(* Logix 5000 project; controller cal1615 1756-L62 rev 20.11; software revision 20.05; part 11 of 82 *)
(* tags used below, declared in another part *)
   FAULT : BOOL;   // Fault AFI
   p00_wac : Accumulator;   // Winder Accumulator
   p01_di_edge_ctrl_estop_active : BOOL;   // System Digital Input Edge Control Estop Active
   p01_di_estop_1_tripped : BOOL;   // System Digital Input EStop Relay 1 Tripped
   p01_di_estop_2_tripped : BOOL;   // System Digital Input EStop Relay 2 Tripped
   p01_di_estop_reset : BOOL;   // System Digital Inupt Main Operator Panel E-Stop Reset
   p01_di_impreg_estop_active : BOOL;   // System Digital Input Impreg Estop Active
   p01_di_letoff_estop_active : BOOL;   // System Digital Input Letoff Estop Active
   p01_di_lof_acc_estop_active : BOOL;   // System Digital Input Letoff Accumulator Estop Active
   p01_di_main_hmi_estop : BOOL;   // System Digital Inupt Main Operator Panel E-Stop Active
   p01_di_rope_sw_1_active : BOOL;   // System Digital Input Rope Switch 1 Active
   p01_di_rope_sw_2_active : BOOL;   // System Digital Input Rope Switch 2 Active
   p01_di_rope_sw_3_active : BOOL;   // System Digital Input Rope Switch 3 Active
   p01_di_rope_sw_4_active : BOOL;   // System Digital Input Rope Switch 4 Active
   p01_di_rope_sw_5_active : BOOL;   // System Digital Input Rope Switch 5 Active
   p01_di_rope_sw_6_active : BOOL;   // System Digital Input Rope Switch 6 Active
   p01_di_rope_sw_7_active : BOOL;   // System Digital Input Rope Switch 7 Active
   p01_di_rope_sw_8_active : BOOL;   // System Digital Input Rope Switch 8 Active
   p01_di_splice_estop_active : BOOL;   // System Digital Input Splice Press Estop Active
   p01_di_ts2_estop_active : BOOL;   // System Digital Input Tension Stand 2 Estop Active
   p01_di_winder_estop_active : BOOL;   // System Digital Input Winder Estop Active
   p01_recipe_active : recipe;   // Active Recipe
   p01r01 : routine;
   p01r02_do_buzzer_LINE : BOOL;
   p01r02_do_green_stack_light_lel : BOOL;   // System Outputs Green Stack Light
   p01r02_do_green_stack_light_LINE : BOOL;
   p01r02_do_red_stack_light : BOOL;   // System Outputs Red Stack Light
   p01r02_do_red_stack_light_LINE : BOOL;
   p01r02_do_yellow_stack_light_LINE : BOOL;
   p01r02_fault_exists : BOOL;
   p01r02_timer_second : TIMER[2];   // System Misc Control Timer Second Pulse
   p01r02_unack_fault : BOOL;   // System Misc Control Unacknowledged Fault Exists
   p01r02_unack_warning : BOOL;   // System Misc Control Unacknowledged Warning Exists
   p01r02_warnings_exists : BOOL;
   p01r04 : routine;   // System Outputs
   p01r09 : routine;   // System Modes
   p01r09_estop_ok : BOOL;   // System Modes Estop Dwell OK
   p01r09_mode_run : BOOL;   // System Modes All Modes Run Mode
   p01r09_open_oven : BOOL;
   p01r09_open_oven_toggle : SYS_Toggle;
   p01r09_pb_global_reset : BOOL;   // System Modes PB: Global Fault Reset
   p01r09_pb_line_jog : BOOL;   // System Modes PB: Line Jog Forward
   p01r09_permissive_change : BOOL;   // System Modes Permissive Mode Change
   p01r09_stretch_mode : BOOL;
   p01r09_timer_estop_reset : TIMER;   // System Modes Estop Reset Dwell
   p01r09_timer_fault : TIMER[20];   // System Modes Fault Delay
   p01r09_timer_global_reset : TIMER;   // System Modes Global Reset Timer
   p01r09_timer_warning : TIMER[4];   // System Modes Warning Delay
   p01r10 : routine;   // System Annunciators
   p01r10_fault_exists : BOOL;
   p01r10_unack_fault : DINT;
   p01r10_unack_fault_ex : BOOL;
   p01r10_unack_warn_ex : BOOL;   // System Annunciators Unacknowledged Warning Exists
   p01r10_unack_warning : DINT;   // System Annunciators Unacknowledged Warning Exists
   p01r10_warning_exists : BOOL;
   p01r12_zero_line_speed : BOOL;   // System Line Accel Decel Control Line Speed at Zero
   p01r13_permissive_drives : BOOL;   // System Line Start Sequence Permissive Drives
   p01r13_permissive_line_run : BOOL;   // System Line Start Sequence Permissive Line Run
   p01r13_state : DINT;   // System Line Start Sequence Sequencer Step
   p01r13_status : DINT;   // System Line Start Sequence Encoded Step
   p02_dint_from_hmi : hmi_dint;
   p11r02_fault_exists : BOOL;
   p11r02_unack_fault : BOOL;   // Zone 1 Misc Control Unacknowledged Fault Exists
   p11r02_unack_warning : BOOL;   // Zone 1 Misc Control Unacknowledged Warning Exists
   p11r02_warning_exists : BOOL;
   p11r30 : routine;   // Zone 1 Temperature Control
   p12r02_fault_exists : BOOL;
   p12r02_unack_fault : BOOL;   // Zone 2 Misc Control Unacknowledged Fault Exists
   p12r02_unack_warning : BOOL;   // Zone 2 Misc Control Unacknowledged Warning Exists
   p12r02_warning_exists : BOOL;
   p12r30 : routine;   // Zone 2 Temperature Control
   p13r02_fault_exists : BOOL;
   p13r02_unack_fault : BOOL;   // Zone 3 Misc Control Unacknowledged Fault Exists
   p13r02_unack_warning : BOOL;   // Zone 3 Misc Control Unacknowledged Warning Exists
   p13r02_warning_exists : BOOL;
   p19r02_fault_exists : BOOL;
   p19r02_unack_warning : BOOL;   // Advanced Cooling Misc Control Unacknowledged Warning
   p19r02_warning_exists : BOOL;
   p20r02_fault_exists : BOOL;
   p20r02_unack_fault : BOOL;   // Letoff Misc Control Unacknowledge Fault Exists
   p20r02_unack_warning : BOOL;   // Letoff Misc Control Unacknowledge Warning Exists
   p20r02_warning_exists : BOOL;
   p21r02_fault_exists : BOOL;
   p21r02_unack_fault : BOOL;   // Splice Press Misc Control Unacknowledged Fault Exists
   p21r02_unack_warning : BOOL;   // Splice Press Misc Control Unacknowledged Warning Exists
   p21r02_warning_exists : BOOL;
   p22r02_fault_exists : BOOL;
   p22r02_unack_fault : BOOL;   // Impreg Pickup Roll Misc Control Unacknowledged Fault Exists
   p22r02_unack_warning : BOOL;   // Impreg Pickup Roll Misc Control Unacknowledged Warning Exists
   p22r02_warning_exists : BOOL;
   p22r09_mode_run : BOOL;   // Tension Stand 1 Modes Run Mode
   p23r02 : routine;   // Impreg Misc Control
   p23r02_fault_exists : BOOL;
   p23r02_unack_fault : BOOL;   // Imperg Misc Control Unackn. Fault Exist
   p23r02_unack_warning : BOOL;   // Impreg Misc Control Unackn. Warning Exist
   p23r02_warning_exists : BOOL;
   p24r02_fault_exists : BOOL;
   p24r02_unack_fault : BOOL;   // Tension Stand 2 Misc Control Unacknowledged Fault Exists
   p24r02_unack_warning : BOOL;   // Tension Stand 2 Misc Control Unacknowledged Warning Exists
   p24r02_warning_exists : BOOL;
   p25r02_fault_exists : BOOL;
   p25r02_unack_fault : BOOL;   // Upper Poly Letoff Misc Control Unacknowledged Fault Exists
   p25r02_unack_warning : BOOL;   // Upper Poly Letoff Misc Control Unacknowledged Warning Exists
   p25r02_warning_exists : BOOL;
   p25r09_mode_run : BOOL;   // Tension Stand 2 Modes Run Mode
   p26r02_fault_exists : BOOL;
   p26r02_unack_fault : BOOL;   // Upper Poly Letoff Misc Control Unacknowledged Fault Exists
   p26r02_unack_warning : BOOL;   // Upper Poly Letoff Misc Control Unacknowledged Warning Exists
   p26r02_warning_exists : BOOL;
   p27r02_fault_exists : BOOL;
   p27r02_unack_fault : BOOL;   // Lower Poly Letoff Misc Control Unacknowledged Fault Exists
   p27r02_unack_warning : BOOL;   // Lower Poly Letoff Misc Control Unacknowledged Warning Exists
   p27r02_warning_exists : BOOL;
   p28r02_fault_exists : BOOL;
   p28r02_unack_fault : BOOL;
   p28r02_unack_warning : BOOL;
   p28r02_warning_exists : BOOL;
   p29r02_fault_exists : BOOL;
   p29r02_unack_fault : BOOL;   // Winder Misc Control Unacknowledged Fault Exists
   p29r02_unack_warning : BOOL;   // Winder Misc Control Unackn. Warning Exists
   p29r02_warning_exists : BOOL;
   p30r02_fault_exists : BOOL;
   p30r02_warning_exists : BOOL;
(* P01_System, continued *)

ROUTINE R09_Modes   (* ladder *)
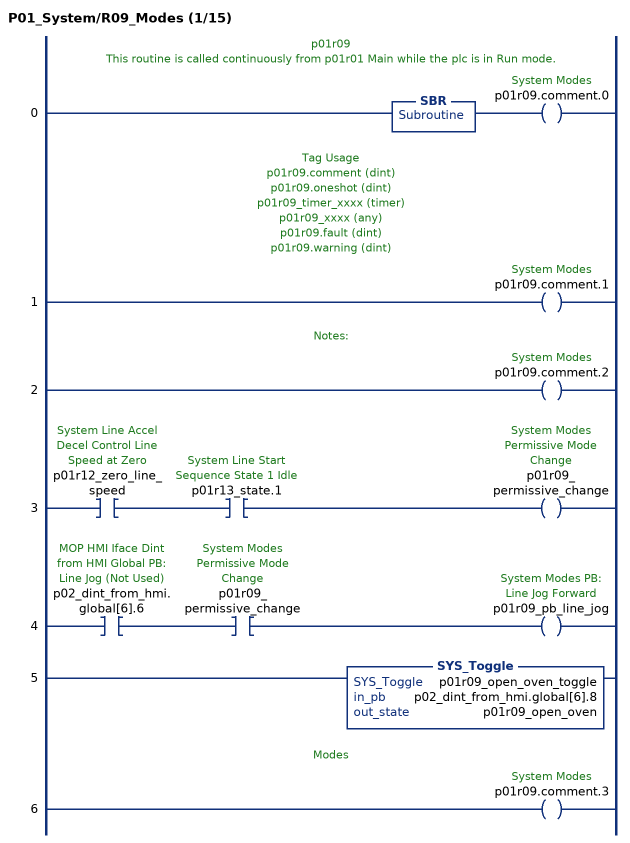
   // p01r09
   // This routine is called continuously from p01r01 Main while the plc is in Run mode.
   0: SBR()OTE(p01r09.comment.0);
   // Tag Usage
   // p01r09.comment (dint)
   // p01r09.oneshot (dint)
   // p01r09_timer_xxxx (timer)
   // p01r09_xxxx (any)
   // p01r09.fault (dint)
   // p01r09.warning (dint)
   1: OTE(p01r09.comment.1);
   // Notes:
   2: OTE(p01r09.comment.2);
   3: XIC(p01r12_zero_line_speed)XIC(p01r13_state.1)OTE(p01r09_permissive_change);
   4: XIC(p02_dint_from_hmi.global[6].6)XIC(p01r09_permissive_change)OTE(p01r09_pb_line_jog);
   5: SYS_Toggle(p01r09_open_oven_toggle,p02_dint_from_hmi.global[6].8,p01r09_open_oven);
   // Modes
   6: OTE(p01r09.comment.3);
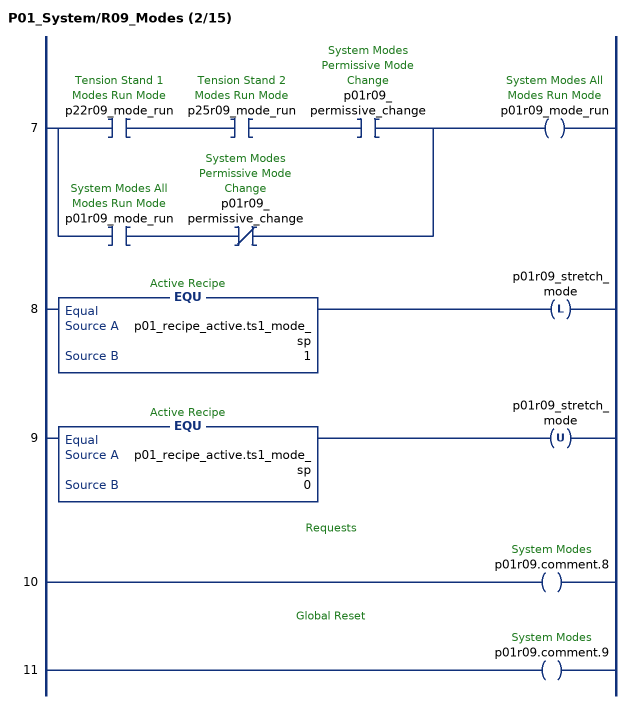
   7: [XIC(p22r09_mode_run) XIC(p25r09_mode_run) XIC(p01r09_permissive_change) ,XIC(p01r09_mode_run) XIO(p01r09_permissive_change) ]OTE(p01r09_mode_run);
   8: EQU(p01_recipe_active.ts1_mode_sp,1)OTL(p01r09_stretch_mode);
   9: EQU(p01_recipe_active.ts1_mode_sp,0)OTU(p01r09_stretch_mode);
   // Requests
   10: OTE(p01r09.comment.8);
   // Global Reset
   11: OTE(p01r09.comment.9);
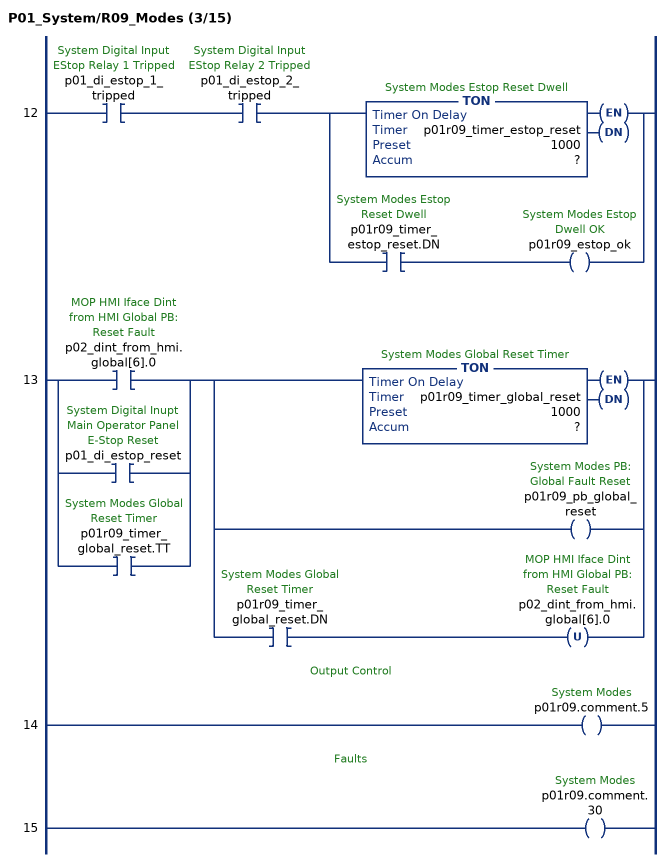
   12: XIC(p01_di_estop_1_tripped)XIC(p01_di_estop_2_tripped)[TON(p01r09_timer_estop_reset,?,?) ,XIC(p01r09_timer_estop_reset.DN) OTE(p01r09_estop_ok) ];
   13: [XIC(p02_dint_from_hmi.global[6].0) ,XIC(p01_di_estop_reset) ,XIC(p01r09_timer_global_reset.TT) ][TON(p01r09_timer_global_reset,?,?) ,OTE(p01r09_pb_global_reset) ,XIC(p01r09_timer_global_reset.DN) OTU(p02_dint_from_hmi.global[6].0) ];
   // Output Control
   14: OTE(p01r09.comment.5);
   // Faults
   15: OTE(p01r09.comment.30);
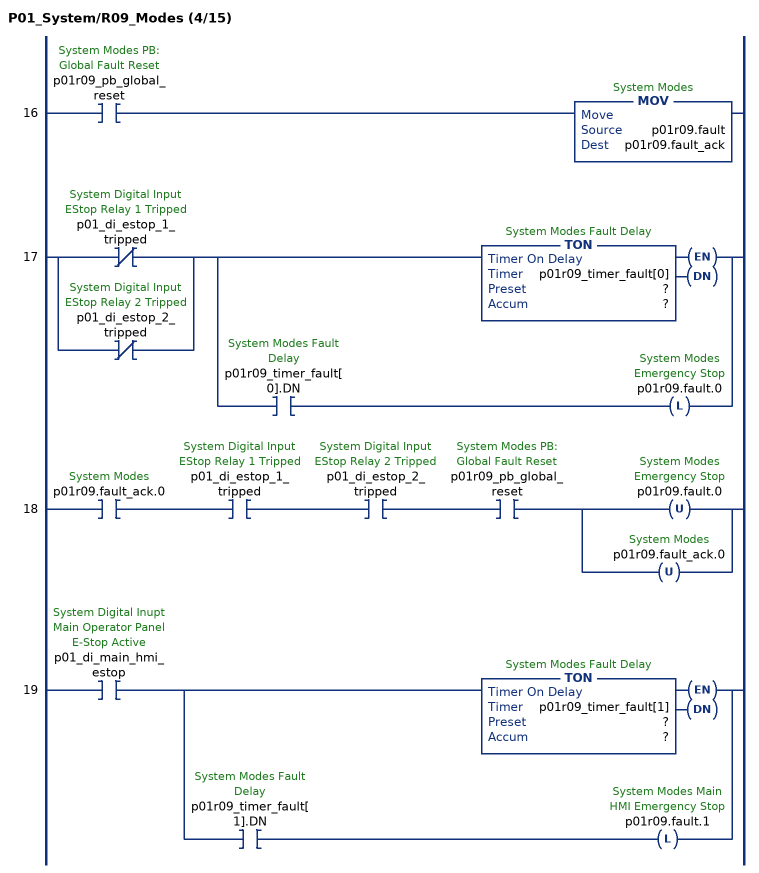
   16: XIC(p01r09_pb_global_reset)MOV(p01r09.fault,p01r09.fault_ack);
   17: [XIO(p01_di_estop_1_tripped) ,XIO(p01_di_estop_2_tripped) ][TON(p01r09_timer_fault[0],?,?) ,XIC(p01r09_timer_fault[0].DN) OTL(p01r09.fault.0) ];
   18: XIC(p01r09.fault_ack.0)XIC(p01_di_estop_1_tripped)XIC(p01_di_estop_2_tripped)XIC(p01r09_pb_global_reset)[OTU(p01r09.fault.0) ,OTU(p01r09.fault_ack.0) ];
   19: XIC(p01_di_main_hmi_estop)[TON(p01r09_timer_fault[1],?,?) ,XIC(p01r09_timer_fault[1].DN) OTL(p01r09.fault.1) ];
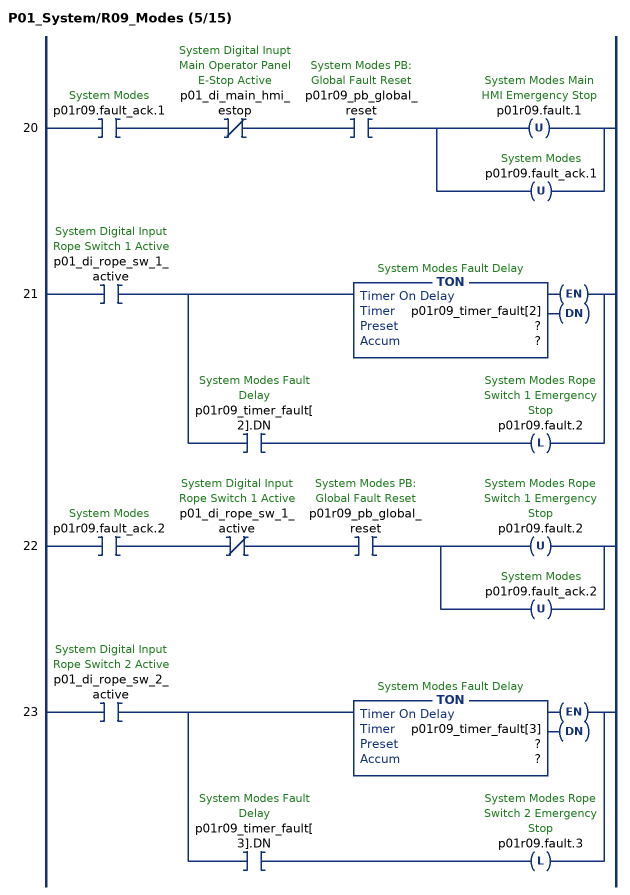
   20: XIC(p01r09.fault_ack.1)XIO(p01_di_main_hmi_estop)XIC(p01r09_pb_global_reset)[OTU(p01r09.fault.1) ,OTU(p01r09.fault_ack.1) ];
   21: XIC(p01_di_rope_sw_1_active)[TON(p01r09_timer_fault[2],?,?) ,XIC(p01r09_timer_fault[2].DN) OTL(p01r09.fault.2) ];
   22: XIC(p01r09.fault_ack.2)XIO(p01_di_rope_sw_1_active)XIC(p01r09_pb_global_reset)[OTU(p01r09.fault.2) ,OTU(p01r09.fault_ack.2) ];
   23: XIC(p01_di_rope_sw_2_active)[TON(p01r09_timer_fault[3],?,?) ,XIC(p01r09_timer_fault[3].DN) OTL(p01r09.fault.3) ];
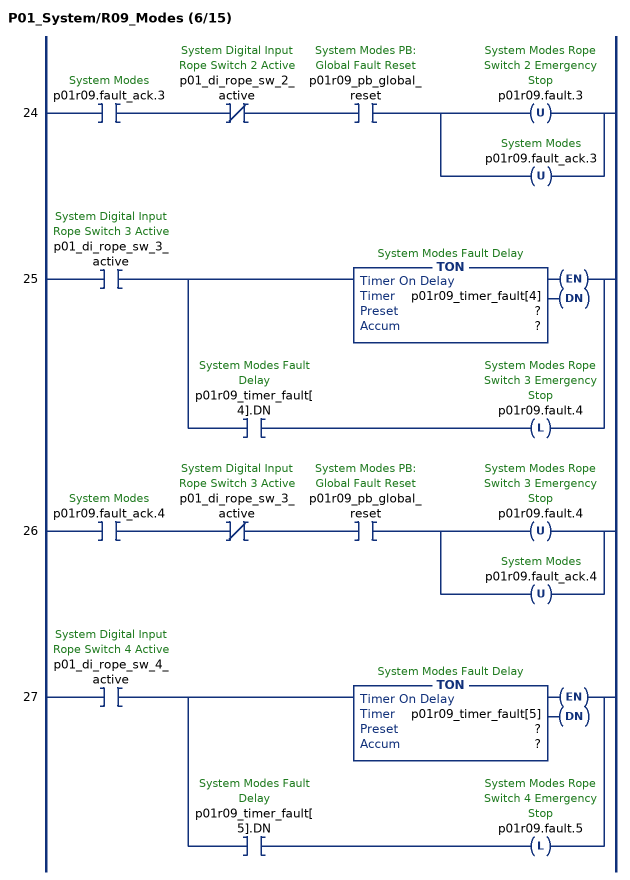
   24: XIC(p01r09.fault_ack.3)XIO(p01_di_rope_sw_2_active)XIC(p01r09_pb_global_reset)[OTU(p01r09.fault.3) ,OTU(p01r09.fault_ack.3) ];
   25: XIC(p01_di_rope_sw_3_active)[TON(p01r09_timer_fault[4],?,?) ,XIC(p01r09_timer_fault[4].DN) OTL(p01r09.fault.4) ];
   26: XIC(p01r09.fault_ack.4)XIO(p01_di_rope_sw_3_active)XIC(p01r09_pb_global_reset)[OTU(p01r09.fault.4) ,OTU(p01r09.fault_ack.4) ];
   27: XIC(p01_di_rope_sw_4_active)[TON(p01r09_timer_fault[5],?,?) ,XIC(p01r09_timer_fault[5].DN) OTL(p01r09.fault.5) ];
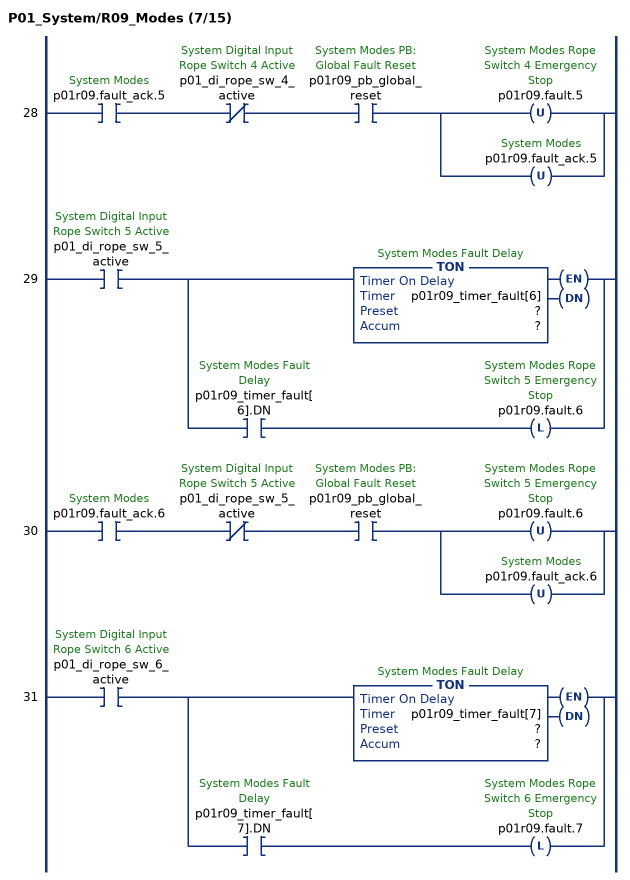
   28: XIC(p01r09.fault_ack.5)XIO(p01_di_rope_sw_4_active)XIC(p01r09_pb_global_reset)[OTU(p01r09.fault.5) ,OTU(p01r09.fault_ack.5) ];
   29: XIC(p01_di_rope_sw_5_active)[TON(p01r09_timer_fault[6],?,?) ,XIC(p01r09_timer_fault[6].DN) OTL(p01r09.fault.6) ];
   30: XIC(p01r09.fault_ack.6)XIO(p01_di_rope_sw_5_active)XIC(p01r09_pb_global_reset)[OTU(p01r09.fault.6) ,OTU(p01r09.fault_ack.6) ];
   31: XIC(p01_di_rope_sw_6_active)[TON(p01r09_timer_fault[7],?,?) ,XIC(p01r09_timer_fault[7].DN) OTL(p01r09.fault.7) ];
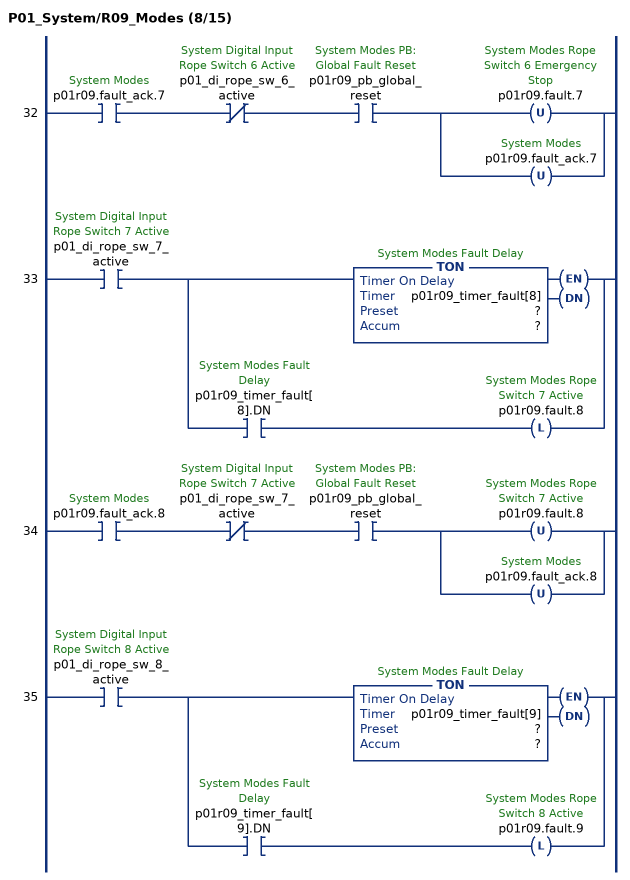
   32: XIC(p01r09.fault_ack.7)XIO(p01_di_rope_sw_6_active)XIC(p01r09_pb_global_reset)[OTU(p01r09.fault.7) ,OTU(p01r09.fault_ack.7) ];
   33: XIC(p01_di_rope_sw_7_active)[TON(p01r09_timer_fault[8],?,?) ,XIC(p01r09_timer_fault[8].DN) OTL(p01r09.fault.8) ];
   34: XIC(p01r09.fault_ack.8)XIO(p01_di_rope_sw_7_active)XIC(p01r09_pb_global_reset)[OTU(p01r09.fault.8) ,OTU(p01r09.fault_ack.8) ];
   35: XIC(p01_di_rope_sw_8_active)[TON(p01r09_timer_fault[9],?,?) ,XIC(p01r09_timer_fault[9].DN) OTL(p01r09.fault.9) ];
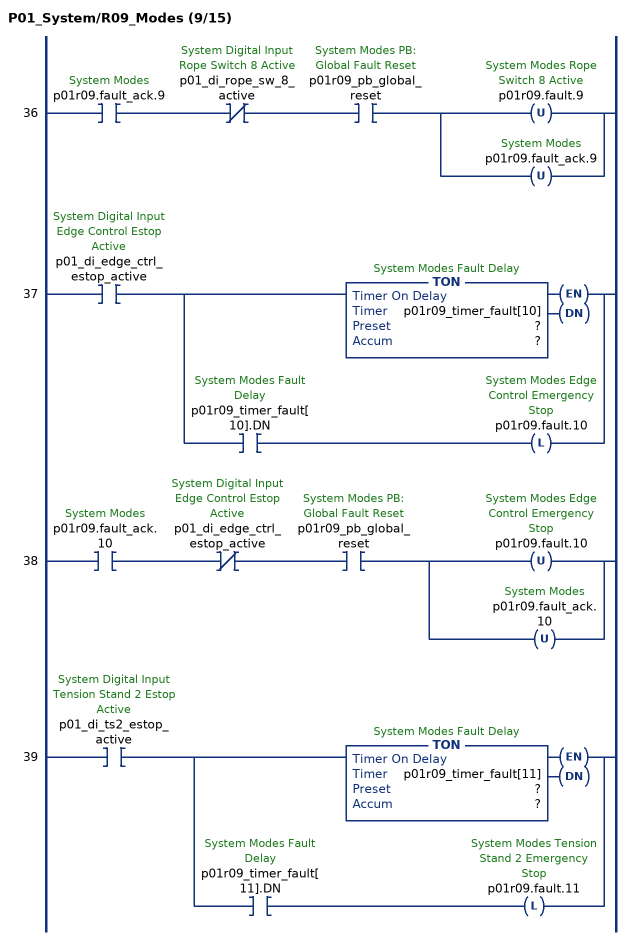
   36: XIC(p01r09.fault_ack.9)XIO(p01_di_rope_sw_8_active)XIC(p01r09_pb_global_reset)[OTU(p01r09.fault.9) ,OTU(p01r09.fault_ack.9) ];
   37: XIC(p01_di_edge_ctrl_estop_active)[TON(p01r09_timer_fault[10],?,?) ,XIC(p01r09_timer_fault[10].DN) OTL(p01r09.fault.10) ];
   38: XIC(p01r09.fault_ack.10)XIO(p01_di_edge_ctrl_estop_active)XIC(p01r09_pb_global_reset)[OTU(p01r09.fault.10) ,OTU(p01r09.fault_ack.10) ];
   39: XIC(p01_di_ts2_estop_active)[TON(p01r09_timer_fault[11],?,?) ,XIC(p01r09_timer_fault[11].DN) OTL(p01r09.fault.11) ];
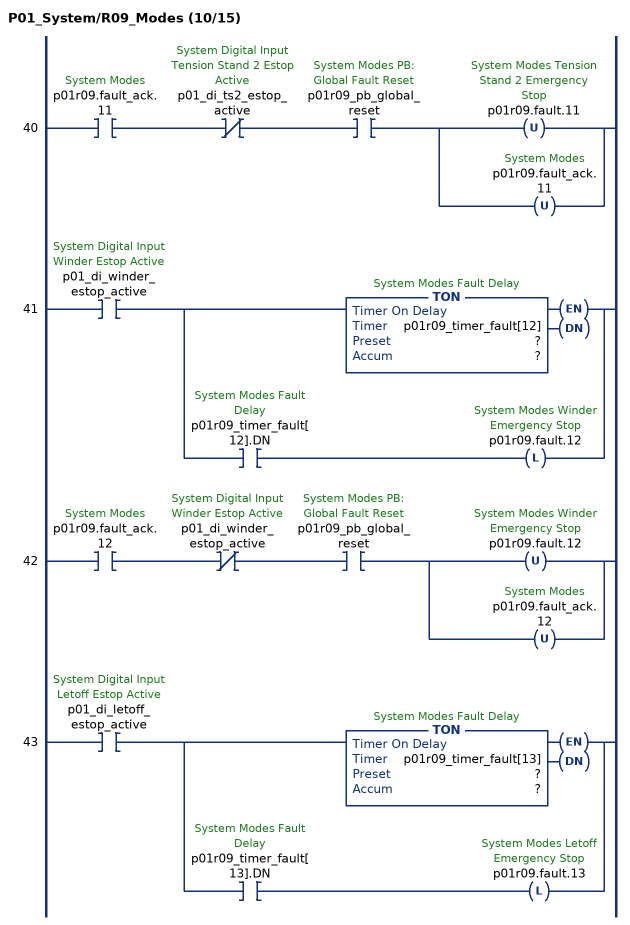
   40: XIC(p01r09.fault_ack.11)XIO(p01_di_ts2_estop_active)XIC(p01r09_pb_global_reset)[OTU(p01r09.fault.11) ,OTU(p01r09.fault_ack.11) ];
   41: XIC(p01_di_winder_estop_active)[TON(p01r09_timer_fault[12],?,?) ,XIC(p01r09_timer_fault[12].DN) OTL(p01r09.fault.12) ];
   42: XIC(p01r09.fault_ack.12)XIO(p01_di_winder_estop_active)XIC(p01r09_pb_global_reset)[OTU(p01r09.fault.12) ,OTU(p01r09.fault_ack.12) ];
   43: XIC(p01_di_letoff_estop_active)[TON(p01r09_timer_fault[13],?,?) ,XIC(p01r09_timer_fault[13].DN) OTL(p01r09.fault.13) ];
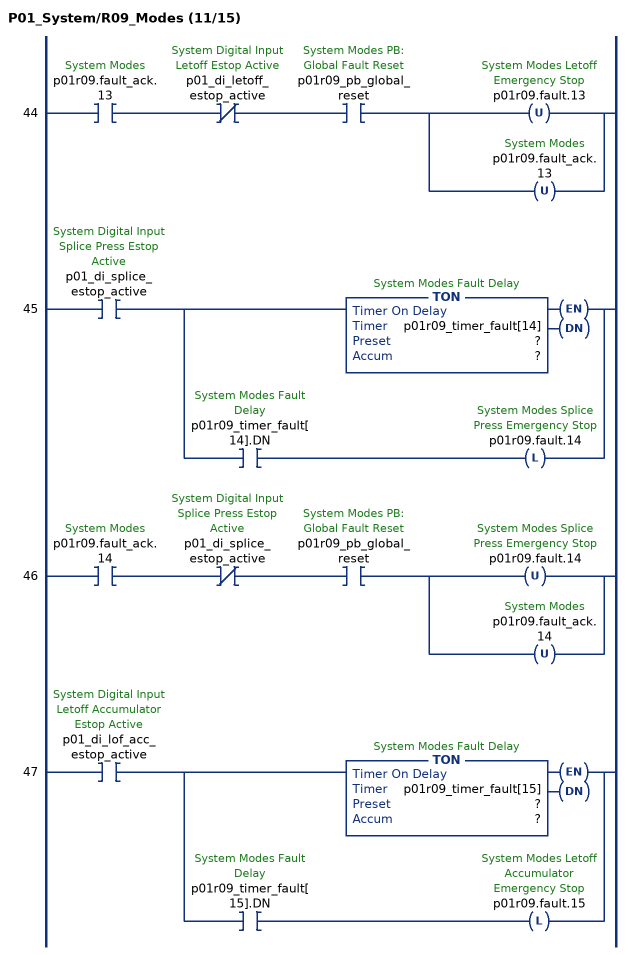
   44: XIC(p01r09.fault_ack.13)XIO(p01_di_letoff_estop_active)XIC(p01r09_pb_global_reset)[OTU(p01r09.fault.13) ,OTU(p01r09.fault_ack.13) ];
   45: XIC(p01_di_splice_estop_active)[TON(p01r09_timer_fault[14],?,?) ,XIC(p01r09_timer_fault[14].DN) OTL(p01r09.fault.14) ];
   46: XIC(p01r09.fault_ack.14)XIO(p01_di_splice_estop_active)XIC(p01r09_pb_global_reset)[OTU(p01r09.fault.14) ,OTU(p01r09.fault_ack.14) ];
   47: XIC(p01_di_lof_acc_estop_active)[TON(p01r09_timer_fault[15],?,?) ,XIC(p01r09_timer_fault[15].DN) OTL(p01r09.fault.15) ];
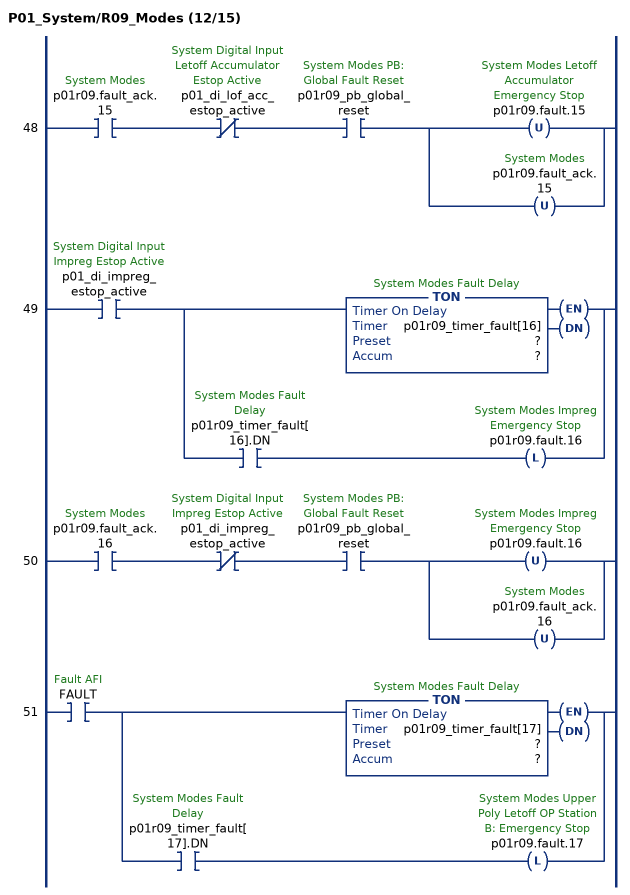
   48: XIC(p01r09.fault_ack.15)XIO(p01_di_lof_acc_estop_active)XIC(p01r09_pb_global_reset)[OTU(p01r09.fault.15) ,OTU(p01r09.fault_ack.15) ];
   49: XIC(p01_di_impreg_estop_active)[TON(p01r09_timer_fault[16],?,?) ,XIC(p01r09_timer_fault[16].DN) OTL(p01r09.fault.16) ];
   50: XIC(p01r09.fault_ack.16)XIO(p01_di_impreg_estop_active)XIC(p01r09_pb_global_reset)[OTU(p01r09.fault.16) ,OTU(p01r09.fault_ack.16) ];
   51: XIC(FAULT)[TON(p01r09_timer_fault[17],?,?) ,XIC(p01r09_timer_fault[17].DN) OTL(p01r09.fault.17) ];
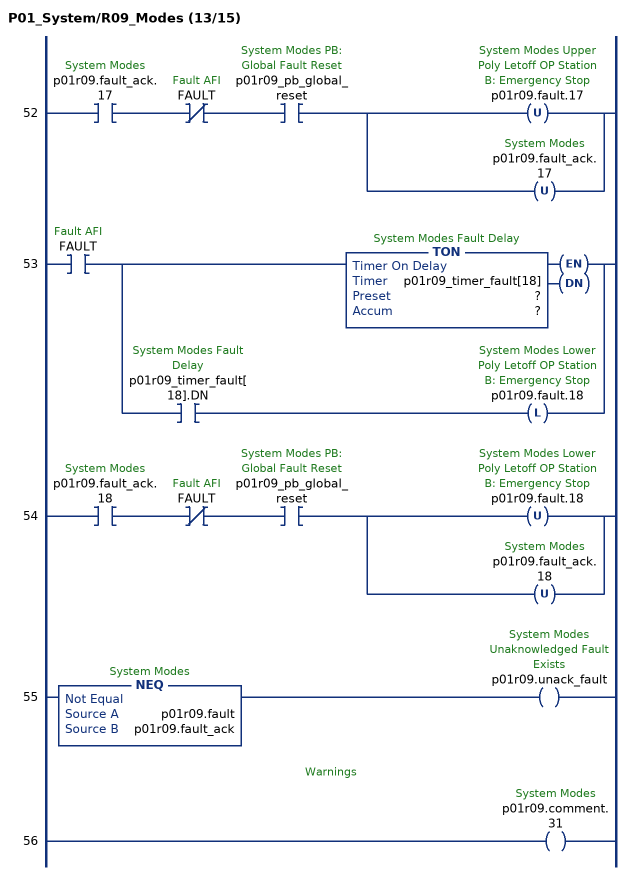
   52: XIC(p01r09.fault_ack.17)XIO(FAULT)XIC(p01r09_pb_global_reset)[OTU(p01r09.fault.17) ,OTU(p01r09.fault_ack.17) ];
   53: XIC(FAULT)[TON(p01r09_timer_fault[18],?,?) ,XIC(p01r09_timer_fault[18].DN) OTL(p01r09.fault.18) ];
   54: XIC(p01r09.fault_ack.18)XIO(FAULT)XIC(p01r09_pb_global_reset)[OTU(p01r09.fault.18) ,OTU(p01r09.fault_ack.18) ];
   55: NEQ(p01r09.fault,p01r09.fault_ack)OTE(p01r09.unack_fault);
   // Warnings
   56: OTE(p01r09.comment.31);
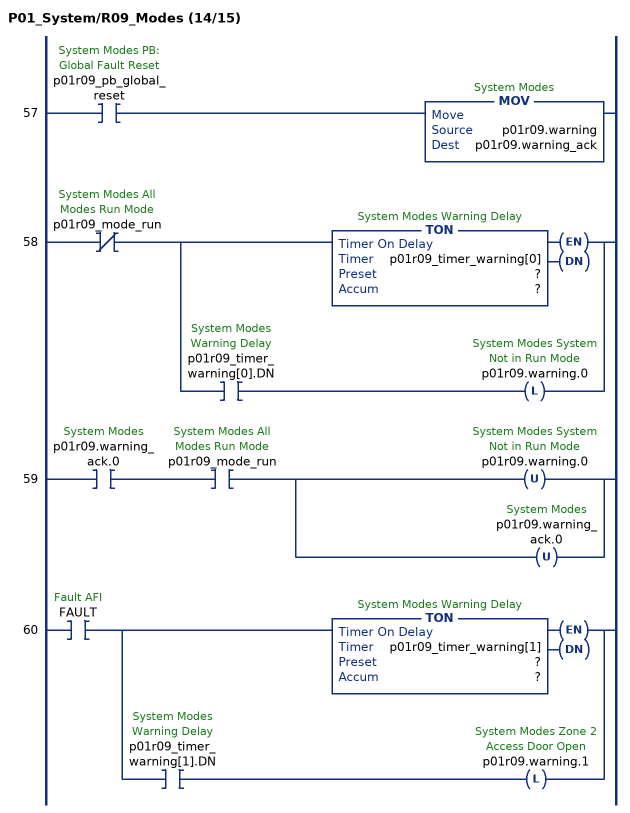
   57: XIC(p01r09_pb_global_reset)MOV(p01r09.warning,p01r09.warning_ack);
   58: XIO(p01r09_mode_run)[TON(p01r09_timer_warning[0],?,?) ,XIC(p01r09_timer_warning[0].DN) OTL(p01r09.warning.0) ];
   59: XIC(p01r09.warning_ack.0)XIC(p01r09_mode_run)[OTU(p01r09.warning.0) ,OTU(p01r09.warning_ack.0) ];
   60: XIC(FAULT)[TON(p01r09_timer_warning[1],?,?) ,XIC(p01r09_timer_warning[1].DN) OTL(p01r09.warning.1) ];
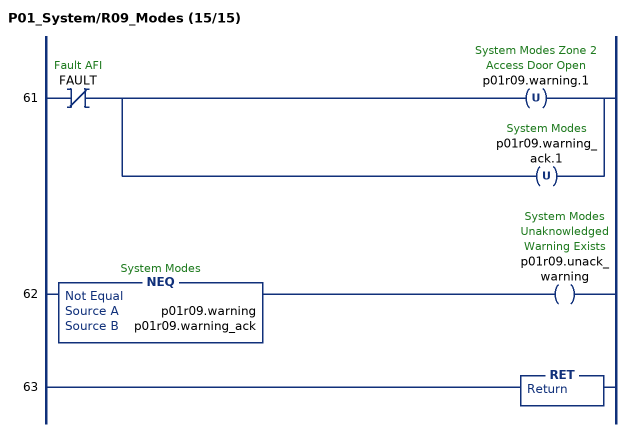
   61: XIO(FAULT)[OTU(p01r09.warning.1) ,OTU(p01r09.warning_ack.1) ];
   62: NEQ(p01r09.warning,p01r09.warning_ack)OTE(p01r09.unack_warning);
   63: RET();
END_ROUTINE

ROUTINE R10_Annunciators   (* ladder *)
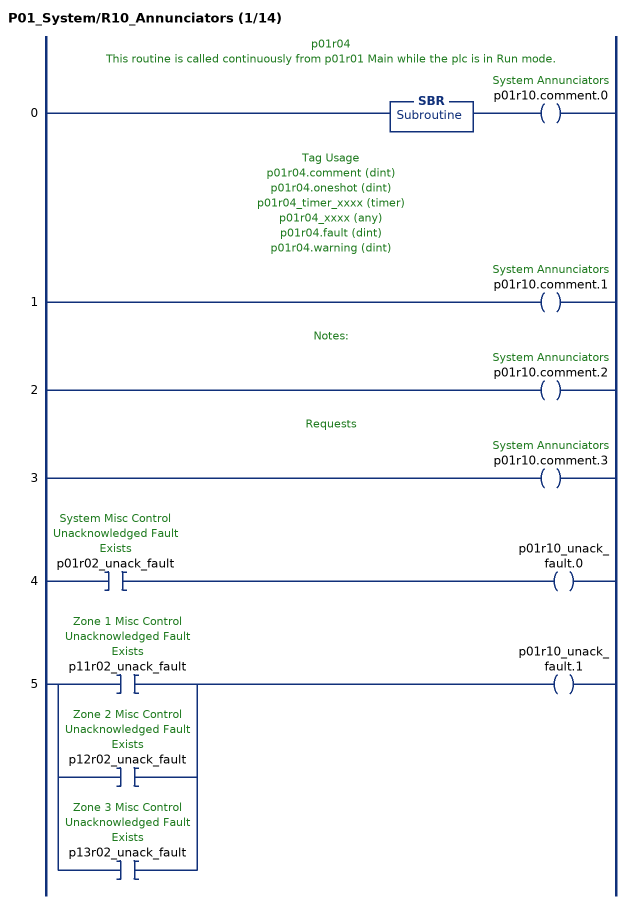
   // p01r04
   // This routine is called continuously from p01r01 Main while the plc is in Run mode.
   0: SBR()OTE(p01r10.comment.0);
   // Tag Usage
   // p01r04.comment (dint)
   // p01r04.oneshot (dint)
   // p01r04_timer_xxxx (timer)
   // p01r04_xxxx (any)
   // p01r04.fault (dint)
   // p01r04.warning (dint)
   1: OTE(p01r10.comment.1);
   // Notes:
   2: OTE(p01r10.comment.2);
   // Requests
   3: OTE(p01r10.comment.3);
   4: XIC(p01r02_unack_fault)OTE(p01r10_unack_fault.0);
   5: [XIC(p11r02_unack_fault) ,XIC(p12r02_unack_fault) ,XIC(p13r02_unack_fault) ]OTE(p01r10_unack_fault.1);
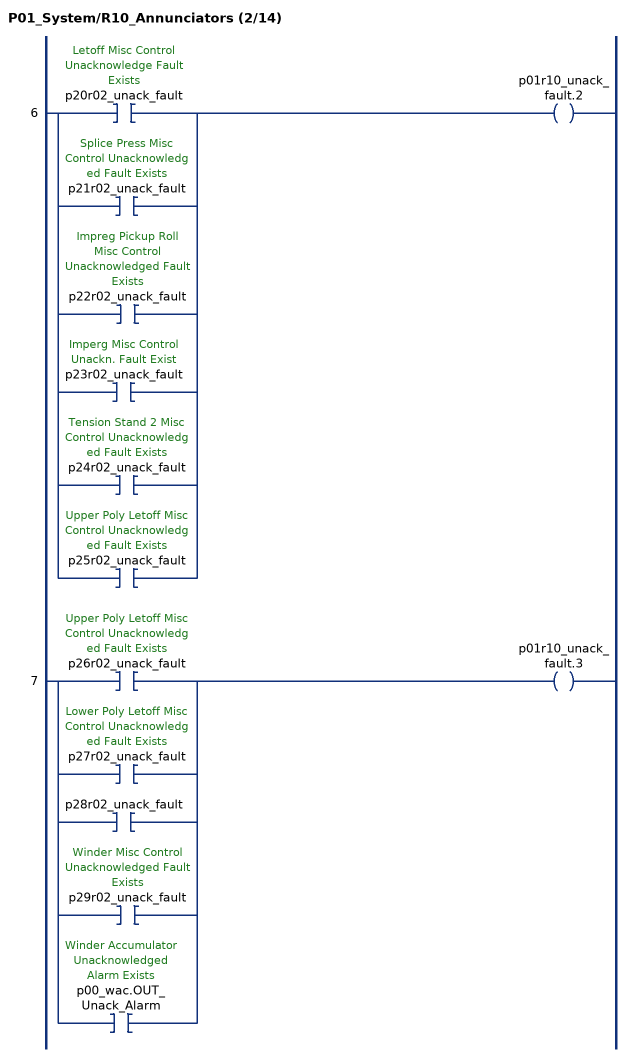
   6: [XIC(p20r02_unack_fault) ,XIC(p21r02_unack_fault) ,XIC(p22r02_unack_fault) ,XIC(p23r02_unack_fault) ,XIC(p24r02_unack_fault) ,XIC(p25r02_unack_fault) ]OTE(p01r10_unack_fault.2);
   7: [XIC(p26r02_unack_fault) ,XIC(p27r02_unack_fault) ,XIC(p28r02_unack_fault) ,XIC(p29r02_unack_fault) ,XIC(p00_wac.OUT_Unack_Alarm) ]OTE(p01r10_unack_fault.3);
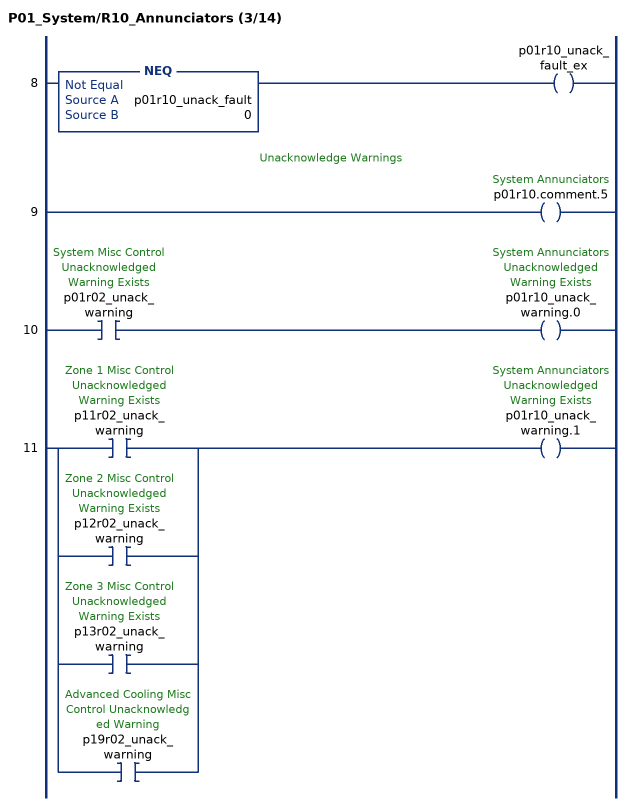
   8: NEQ(p01r10_unack_fault,0)OTE(p01r10_unack_fault_ex);
   // Unacknowledge Warnings
   9: OTE(p01r10.comment.5);
   10: XIC(p01r02_unack_warning)OTE(p01r10_unack_warning.0);
   11: [XIC(p11r02_unack_warning) ,XIC(p12r02_unack_warning) ,XIC(p13r02_unack_warning) ,XIC(p19r02_unack_warning) ]OTE(p01r10_unack_warning.1);
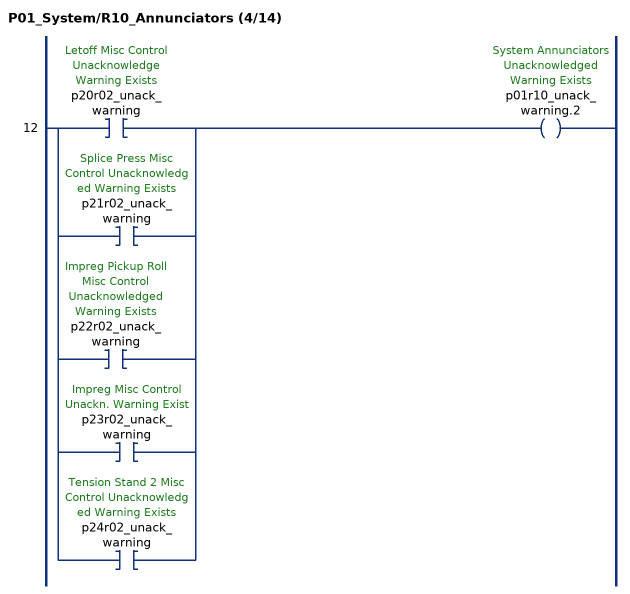
   12: [XIC(p20r02_unack_warning) ,XIC(p21r02_unack_warning) ,XIC(p22r02_unack_warning) ,XIC(p23r02_unack_warning) ,XIC(p24r02_unack_warning) ]OTE(p01r10_unack_warning.2);
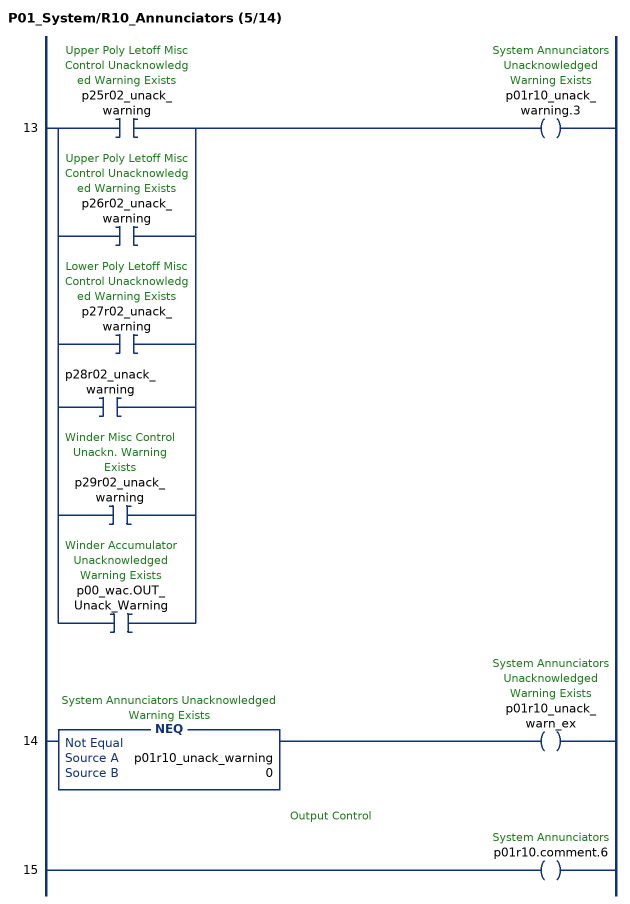
   13: [XIC(p25r02_unack_warning) ,XIC(p26r02_unack_warning) ,XIC(p27r02_unack_warning) ,XIC(p28r02_unack_warning) ,XIC(p29r02_unack_warning) ,XIC(p00_wac.OUT_Unack_Warning) ]OTE(p01r10_unack_warning.3);
   14: NEQ(p01r10_unack_warning,0)OTE(p01r10_unack_warn_ex);
   // Output Control
   15: OTE(p01r10.comment.6);
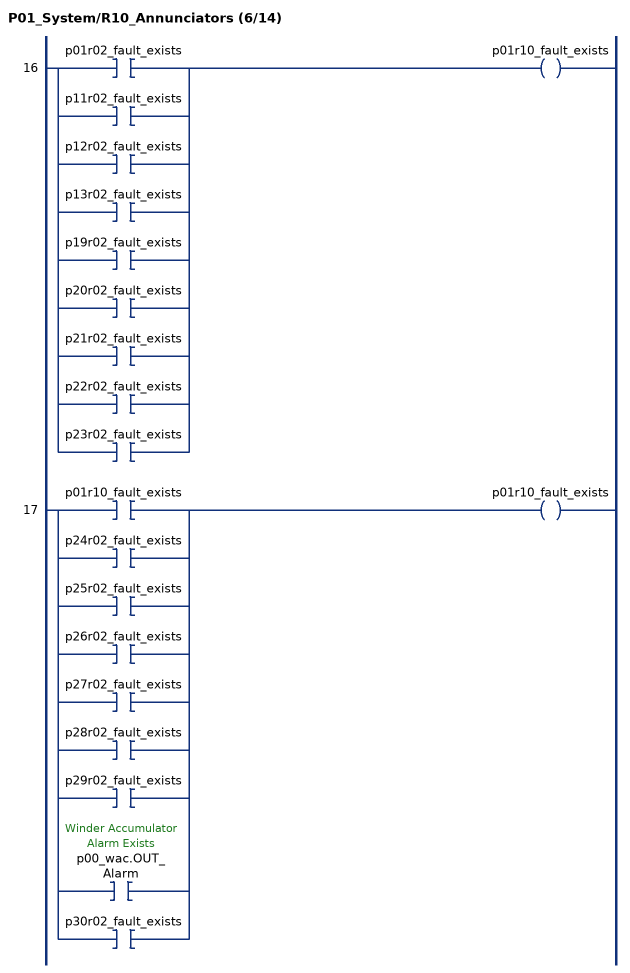
   16: [XIC(p01r02_fault_exists) ,XIC(p11r02_fault_exists) ,XIC(p12r02_fault_exists) ,XIC(p13r02_fault_exists) ,XIC(p19r02_fault_exists) ,XIC(p20r02_fault_exists) ,XIC(p21r02_fault_exists) ,XIC(p22r02_fault_exists) ,XIC(p23r02_fault_exists) ]OTE(p01r10_fault_exists);
   17: [XIC(p01r10_fault_exists) ,XIC(p24r02_fault_exists) ,XIC(p25r02_fault_exists) ,XIC(p26r02_fault_exists) ,XIC(p27r02_fault_exists) ,XIC(p28r02_fault_exists) ,XIC(p29r02_fault_exists) ,XIC(p00_wac.OUT_Alarm) ,XIC(p30r02_fault_exists) ]OTE(p01r10_fault_exists);
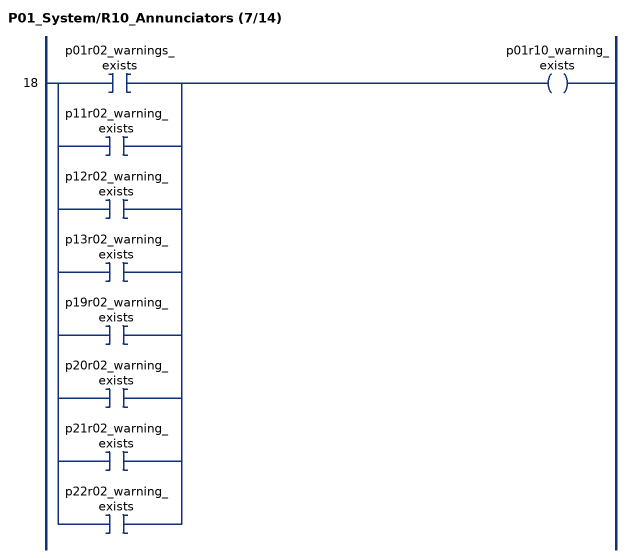
   18: [XIC(p01r02_warnings_exists) ,XIC(p11r02_warning_exists) ,XIC(p12r02_warning_exists) ,XIC(p13r02_warning_exists) ,XIC(p19r02_warning_exists) ,XIC(p20r02_warning_exists) ,XIC(p21r02_warning_exists) ,XIC(p22r02_warning_exists) ]OTE(p01r10_warning_exists);
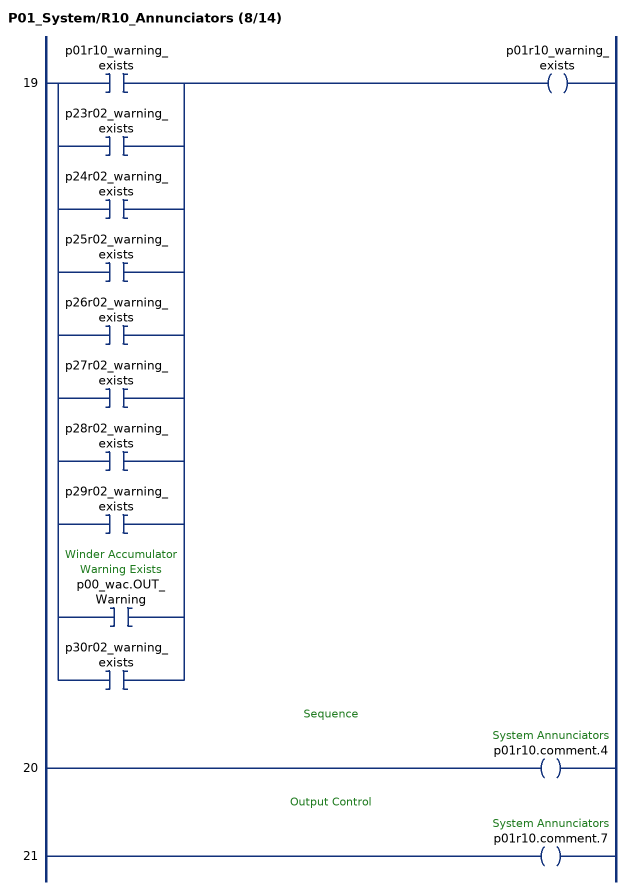
   19: [XIC(p01r10_warning_exists) ,XIC(p23r02_warning_exists) ,XIC(p24r02_warning_exists) ,XIC(p25r02_warning_exists) ,XIC(p26r02_warning_exists) ,XIC(p27r02_warning_exists) ,XIC(p28r02_warning_exists) ,XIC(p29r02_warning_exists) ,XIC(p00_wac.OUT_Warning) ,XIC(p30r02_warning_exists) ]OTE(p01r10_warning_exists);
   // Sequence
   20: OTE(p01r10.comment.4);
   // Output Control
   21: OTE(p01r10.comment.7);
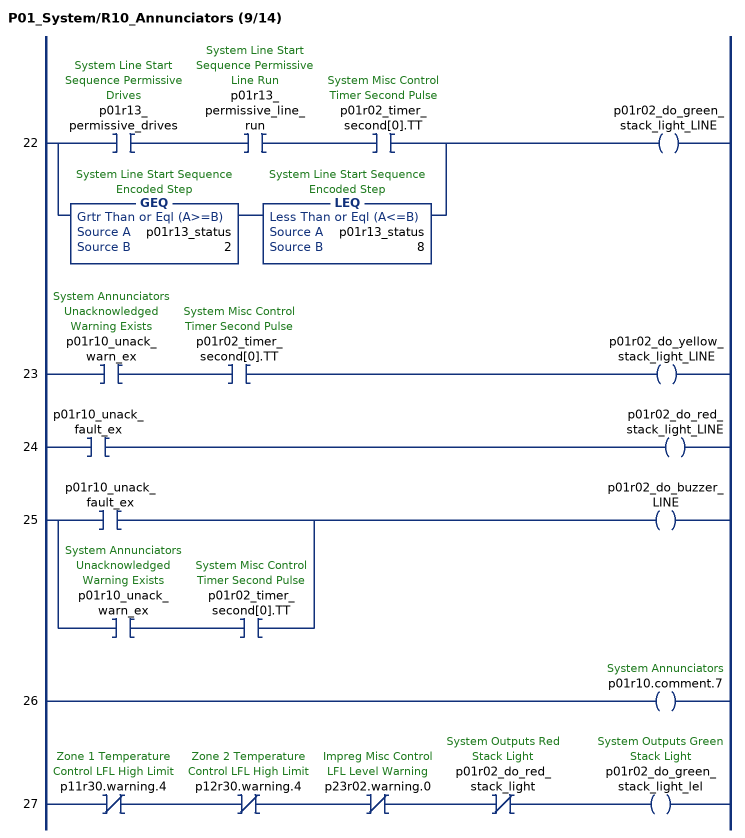
   22: [XIC(p01r13_permissive_drives) XIC(p01r13_permissive_line_run) XIC(p01r02_timer_second[0].TT) ,GEQ(p01r13_status,2) LEQ(p01r13_status,8) ]OTE(p01r02_do_green_stack_light_LINE);
   23: XIC(p01r10_unack_warn_ex)XIC(p01r02_timer_second[0].TT)OTE(p01r02_do_yellow_stack_light_LINE);
   24: XIC(p01r10_unack_fault_ex)OTE(p01r02_do_red_stack_light_LINE);
   25: [XIC(p01r10_unack_fault_ex) ,XIC(p01r10_unack_warn_ex) XIC(p01r02_timer_second[0].TT) ]OTE(p01r02_do_buzzer_LINE);
   26: OTE(p01r10.comment.7);
   27: XIO(p11r30.warning.4)XIO(p12r30.warning.4)XIO(p23r02.warning.0)XIO(p01r02_do_red_stack_light)OTE(p01r02_do_green_stack_light_lel);
